// TwinCAT 3 PLC project Untitled1
// ProgramVersion: 3.1.4026.19
// libraries:
//   Tc2_Standard, * (Beckhoff Automation GmbH)
//   Tc2_System, * (Beckhoff Automation GmbH)
//   Tc2_Utilities, * (Beckhoff Automation GmbH)
//   Tc3_EventLogger, * (Beckhoff Automation GmbH)
//   Tc3_Module, * (Beckhoff Automation GmbH)
// project tree:
//   DUTs/ FlexChain.TcDUT, E_LightStates.TcDUT, E_SwitchType.TcDUT (not stored)
//   FaultChecker/ E_EventType.TcDUT, FB_EventTrigger.TcPOU, TriggerData.TcDUT, TC_EventSeverityToString.TcPOU, TriggerSettings.TcDUT
//   GVLs/ GVL_Fault.TcGVL, GVL_IO.TcGVL
//   Junk/ CdEventSeverity.TcTLEO, E_MachineStatus.TcDUT, FB_FaultChecker.TcPOU
//   / PlcTask.TcTTO
//   POUs/ fbDigitalInput.TcPOU, DigitalIO.TcPOU, fbDigitalOutput.TcPOU, MAIN.TcPOU
//   POUs/Hardware/PULS PISA/DTUs/ CircuitBreakerStatus.TcTLEO, PisaPulseCommMode.TcTLEO, PISA_HMI.TcDUT, PISA_IO.TcDUT, PulsPisaChannelCount.TcTLEO, TimedPulse.TcDUT
//   POUs/Hardware/PULS PISA/POUs/ FB_PISA.TcPOU, NTP.TcPOU
// real-time tasks:
//   TASK PlcTask: cycle T#2ms, priority 20, ADS port 350
// I/O:
//   DEVICE Device 1 (EtherCAT) (disabled), AmsNetId 10.1.14.1.2.1
//     Term 7 (EK1200)
//     Box 12 (Flexi Gateway GETC1)
//     Box 13 (EP6228-0022)
//   DEVICE Device 2 (EtherCAT), AmsNetId 0.0.0.0.3.1
//     Box 1 (EP6228-0022) [EP6228-0022 (IO Link Master)]
//       modules: Module 1 (DeviceState Inputs Device), Module 2 (DeviceState Inputs), Module 3 (empty), Module 4 (empty), Module 5 (empty), Module 6 (empty), Module 7 (empty), Module 8 (empty), Module 9 (empty), Module 10 (IO-Link Slave)
// variable links:
//   Untitled1/Untitled1 Instance <-> Device 1 (EtherCAT)/Box 13 (EP6228-0022)
//     PlcTask Inputs/GVL_IO.Encoder_Counts <-> Module 3 (IO-Link Slave)/IO-Link Port1/Counter
//     PlcTask Inputs/GVL_IO.flexChain.pdo[0] <-> Module 4 (IO-Link Slave)/IO-Link Port2_in/Process Data In
//     PlcTask Inputs/GVL_IO.flexChain.pdo[{1..12}] <-> Module 4 (IO-Link Slave)/IO-Link Port2_in/Process Data In_{1..12}  (12 links)
//   Untitled1/Untitled1 Instance <-> Device 1 (EtherCAT)/Term 7 (EK1200)/Term 10 (EL2008)
//     PlcTask Outputs/GVL_IO.aOutputs[1] <-> Channel 1/Output
//     PlcTask Outputs/GVL_IO.aOutputs[2] <-> Channel 2/Output
//   Untitled1/Untitled1 Instance <-> Device 1 (EtherCAT)/Term 7 (EK1200)/Term 9 (EL1008)
//     PlcTask Inputs/GVL_IO.aInputs[1] <-> Channel 1/Input
//     PlcTask Inputs/GVL_IO.aInputs[2] <-> Channel 2/Input
//     PlcTask Inputs/GVL_IO.aInputs[8] <-> Channel 8/Input
//   Untitled1/Untitled1 Instance <-> Device 2 (EtherCAT)/Box 1 (EP6228-0022)
//     PlcTask Inputs/MAIN.myPisa.PisaIO.bRX <-> Module 10 (IO-Link Slave)/IO-Link Port8_in/DI [X1.6-2] (pin 2)
//     PlcTask Outputs/MAIN.myPisa.PisaIO.bTX <-> Module 10 (IO-Link Slave)/IO-Link Port8_out/DO [X1.6-1] (pin 4)

CONFIGURATION Untitled1
    RESOURCE PLC ON TwinCAT3
        TASK PlcTask(INTERVAL := T#2ms, PRIORITY := 20);
        PROGRAM MAIN WITH PlcTask : MAIN;
    END_RESOURCE
END_CONFIGURATION

// ---- DUTs/FlexChain.TcDUT
TYPE FlexChain :
STRUCT
	pdo AT %I* : ARRAY[0..31] OF BYTE;//max pdo inputs of the flex chain bus
END_STRUCT
END_TYPE

// ---- DUTs/E_LightStates.TcDUT
{attribute 'qualified_only'}
{attribute 'strict'}
TYPE E_LightStates :
(
	OFF := 3,
	ON := 1,
	SLOW_BLINK := 2,
	FAST_BLINK := 0,
	
	
	COUNT  //Max value. Insert new values before to keep this as the max. Used to get max enum size when useful as an input to other function blocks.  
);
END_TYPE

// ---- FaultChecker/E_EventType.TcDUT
{attribute 'qualified_only'}
{attribute 'strict'}
{attribute 'to_string'}
TYPE E_EventType :
(
	Message := 0,
	Alarm :=1
);
END_TYPE

// ---- FaultChecker/TriggerData.TcDUT
TYPE TriggerData :
STRUCT
	nActivationCount: UDINT := 0;
	bTriggered : BOOL;
	
	GetEventTrigger : R_TRIG;
		

	timerDebounceTimer :TON;
	



	
	SendEventTrigger : R_TRIG;

END_STRUCT
END_TYPE

// ---- FaultChecker/TriggerSettings.TcDUT
TYPE TriggerSettings :
STRUCT
	//Settings
	tDebounceTime: TIME :=T#0S;
	nActivationThreshold: UDINT:=1;
	bAutoResetCount: BOOL :=TRUE;
	eEventType :E_EventType:=E_EventType.Message;
END_STRUCT
END_TYPE

// ---- Junk/CdEventSeverity.TcTLEO
{attribute 'qualified_only'}
{attribute 'strict'}
{attribute 'to_string'}
TYPE CdEventSeverity :
(
    Verbose:=0,     // Useful Information for debugging 
    Info:=1,        // Useful Information for operators
    Warning:=2,     // Machine operation not inhibited but at risk of becoming so
    Error:=3,       // Component operation blocked till resolved
    Critical:=4,    // Machine operation bloced till resolved
	                // 5-7 Reserved for future implementaion
	Lockout:=8      // Mackine locked out from use until ADMIN clears Fault 
					// 9 Reserved for future implementaion 
	
);
END_TYPE
//  Lockout = '8      '

// ---- Junk/E_MachineStatus.TcDUT
//{attribute 'qualified_only'}
//{attribute 'strict'}
{attribute 'to_string'}


(*
  |  1---    |  -2---   |  --3-    |   ---4   |  
 -+----------+----------+----------+----------+
0 | System   | Verbose  |    #     |     #    |
1 | Saftey   | Info     |    #     |     #    |
2 | Motor    | Warning  |    #     |     #    |
3 | Air      | Error    |    #     |     #    |
4 | Jam      | Critical |    #     |     #    |
5 | Heat     |          |    #     |     #    |
6 | Reject   |          |    #     |     #    |
7 | Fold     |          |    #     |     #    |
8 | Conveyor | Lockout  |    #     |     #    |
9 | General  |          |    #     |     #    |
  +----------+----------+----------+----------+
*)



TYPE E_MachineStatus:
(
	None                                := 0000,
	//System 0000-0999
	System_Standby		                := 0100,
	System_Running		                := 0101,
    System_Paused 		                := 0102,
	System_VFD_FirmwareUpdate           := 0199,
	Test_Mode           			    := 0104,
	Maintenance_Mode 	                := 0105,
	JogReverse 			                := 0106,
	System_FileError	                := 0400,
	
	//Safety 1000-1999	
	Reset_Safety	                    := 1101,	
	Safety_Fault	                    := 1401,
	Safety_System_Error	                := 1402,
	
	//Saftey - E-STOP XX10-XX19
	EStop_Triggered                     := 1410,
	Front_Left_ES                       := 1411,
	Front_Right_ES                      := 1412,
	Rear_Left_ES                        := 1413,
	Rear_Right_ES                       := 1414,
	External_ES                         := 1415,
	EStop_FB_Fault                     	:= 1419,
	
	//Saftey - Door XX20-XX29
	DoorOpen	                        := 1420,
	Top_Left_Door                       := 1421,
	Top_Right_Door                      := 1422,
	Left_Door                           := 1423,
	Right_Door                          := 1424,
	Rear_Door                           := 1425,
	Front_Panel                         := 1426,
	Door_FB_Fault                       := 1429,
	
	//Motor Fault 2000-2999	
	Skis_Calibrating                    := 2111,
	Motor_Fault	                        := 2450,
	VFD_Primary_Fault                   := 2451,
	VFD_XF1_Fault                       := 2452,
	VFD_XF2_Fault                       := 2453,
	VFD_Stacker_Fault                   := 2454,
	Inlet_Fault                         := 2455,
	Ski_Fault                           := 2456,
	Exit_1_Fault                        := 2461,
	Exit_2_Fault                        := 2462,
	Exit_3_Fault		                := 2463,
	Exit_4_Fault                        := 2464,
	Side_Conveyor_Fault                 := 2470,
	Side_Incline_Fault                  := 2471,
	Side_Conveyor_Unplugged             := 2472,
	
	VFD_Primary_Voltage_Loss            := 2180,
	VFD_XF1_Voltage_Loss                := 2181,
	VFD_XF2_Voltage_Loss                := 2182,
	VFD_Stacker_Voltage_Loss            := 2183,
	VFD_MultipleVoltage_Loss            := 2184,
	
	//Air Status 3000-3999	
	LowAirPressure	                    := 3120,
	HighAirWarning                      := 3221,
	LowAirWarning                       := 3220,
	Filter_Cleaning_Required            := 3333,
	
	//Jam Status 4000-4999	
	Jam_Detected		                := 4400,
	Jam_Inlet                           := 4401,
	Jam_Primary                         := 4402,
	Jam_XF1                             := 4403,
	Jam_XF2                             := 4404,
	Jam_XF2_SensorTimeout               := 4405,
	Jam_Stacker                         := 4406,
	Jam_Stacker_SensorTimeout           := 4407,
	Jam_Stacker_Lane1                   := 4408,
	Jam_Stacker_Lane2                   := 4409,
	Jam_Stacker_Lane3                   := 4410,	
	Jam_Stacker_Lane4                   := 4411,
	Jam_Reject_Rear                     := 4412, 	
	Jam_Reject_Front                    := 4413,
	Jam_Measure_Sensor                  := 4414,
	
	Jam_OverTorquePrimary               := 4415,
	Jam_OverTorqueXF1                   := 4416,
	Jam_OverTorqueXF2                   := 4417,
	Jam_OverTorqueStacker               := 4418,

	//Reject 6000-6999
	//Reject - USER XX00-XX09
	User_Reject                         := 6100,
	User_Reject_Damage                  := 6101,
	User_Reject_Tear  			        := 6102,
	User_Reject_Feed					:= 6103,
	User_Reject_Stain                   := 6104,
	//Reject - Auto XX10-xx40
	Auto_Reject_Unknown                 := 6111,
	OverWideL_Reject                    := 6112,
	OverWideR_Reject                    := 6113,
	Auto_Reject_TooNarrow               := 6114,
	Auto_Reject_TooWide                 := 6115,
	Auto_Reject_TooShort                := 6116,
	Auto_Reject_TooLong                 := 6117,
	Auto_Reject_WrongWidth              := 6118,
	Auto_Reject_WrongLength             := 6119,
	Auto_Reject_XF2_Timeout             := 6121,
	Auto_Reject_ConvLockout             := 6122,
	Auto_Reject_WrongSort               := 6123,
	Auto_Reject_Primary                 := 6124,
	Auto_Reject_Primary_NoSortNum       := 6125,
	Auto_Reject_Crossfold_1             := 6126,
	Auto_Reject_Crossfold_2             := 6127,
	Auto_Reject_Stacker                 := 6128,
	Reject_Unknown	                    := 6129,
		
	//Conveyor	
	Side_Conv_Full                      := 8102,
	Side_Conv_Top_Full 	                := 8103,
	
	//General
	Verbose                             := 9100,
	Info                                := 9200,
	Warning                             := 9300,
	Error                               := 9400,
	Critical                            := 9500,
	Lockout                             := 9800,
	//General - Circuit Breaker XX11-XX19
	Circuit_Breaker_Tripped             := 9411,
	Circuit_Breaker_Tripped_Repeat		:= 9421,
	Circuit_Breaker_Comms_Loss          := 9311,

	//General - SensorAllignment XX20-xx40
	MeasureSensorAlign	                := 9220,
	OverwideLSensorAlign                := 9221,				
	OverwideRSensorAlign                := 9222,
	XF1SensorAlign                      := 9223,
	XF2SensorAlign                      := 9224,
	Stack1SensorAlign                   := 9225, 
	Stack2SensorAlign                   := 9226,
	Stack3SensorAlign                   := 9227,
	Stack4SensorAlign                   := 9228,
	Sort1SensorAlign                    := 9229,
	Sort2SensorAlign                    := 9230,
	Sort3SensorAlign                    := 9231,
	Sort4SensorAlign                    := 9232,	
	Reserved                            := 9999//Leave as last so there aren't compile errors when copy pasting comma seperated values.
)INT;
END_TYPE

// ---- POUs/Hardware/PULS PISA/DTUs/CircuitBreakerStatus.TcTLEO
{attribute 'qualified_only'}
{attribute 'strict'}
TYPE CircuitBreakerStatus :
(
	OFF        := 0, // Channel has been set OFF either manually or programatically (only available in bidirectional mode)
	ON         := 1, // Channel is ON and funcioning normally (only available in bidirectional mode)
	TRIPPED    := 2, // An overcurrent event has tripped the device
	RESET      := 3, // A reset signal has been sent to the device but it hasn't responded yet
	UNKNOWN    := 4, // Comms isssue, data not yet recived, 
	NOTTRIPPED := 5  // Channel is OFF or ON (only available in unidirectional mode)  
);
END_TYPE

// ---- POUs/Hardware/PULS PISA/DTUs/PisaPulseCommMode.TcTLEO
{attribute 'qualified_only'}
{attribute 'strict'}
TYPE PisaPulseCommMode :
(
	Offline :=0,
	Unidirectional := 1,
	Bidirectional :=2
	
);
END_TYPE

// ---- POUs/Hardware/PULS PISA/DTUs/PISA_HMI.TcDUT
TYPE PISA_HMI :
STRUCT
	sCommMode : PisaPulseCommMode := PisaPulseCommMode.Offline;	
	//Variables for Reading
	aStatus : ARRAY[1..8] OF CircuitBreakerStatus := [8(CircuitBreakerStatus.UNKNOWN)];
	aTargetStatus : ARRAY[1..8] OF CircuitBreakerStatus := [8(CircuitBreakerStatus.UNKNOWN)];
END_STRUCT
END_TYPE

// ---- POUs/Hardware/PULS PISA/DTUs/PISA_IO.TcDUT
TYPE PISA_IO :
STRUCT
	sProductName  :STRING;
	bRX AT %I* : BIT;//INPUTS (STATUS -3.4)
	bTX AT %Q* : BIT;//OUTPUTS (CTRL +3.1)
END_STRUCT
END_TYPE

// ---- POUs/Hardware/PULS PISA/DTUs/PulsPisaChannelCount.TcTLEO
{attribute 'qualified_only'}
{attribute 'strict'}
TYPE PulsPisaChannelCount :
(
	FOUR := 4,
	EIGHT :=8
);
END_TYPE

// ---- POUs/Hardware/PULS PISA/DTUs/TimedPulse.TcDUT
TYPE TimedPulse :
STRUCT
	tLeadingGap: TIME   := T#0MS;
	tHighSignal: TIME := T#0MS;
	tTrailingGap: TIME:= T#0MS;
END_STRUCT
END_TYPE

// ---- GVLs/GVL_Fault.TcGVL
{attribute 'qualified_only'}
VAR_GLOBAL
	fbEventTrigger : FB_EventTrigger(TC_EVENT_CLASSES.TestEventClass); 
END_VAR

// ---- GVLs/GVL_IO.TcGVL
{attribute 'qualified_only'}

VAR_GLOBAL CONSTANT
    lightBarPDOstartIndex     : INT := 5;
    lightBarPDOsecondIndex : INT := lightBarPDOstartIndex+1;
END_VAR
VAR_GLOBAL
		Encoder_Counts AT %I* : UINT;
		
		byteArray AT %I* : ARRAY[1..8] OF BOOL;
		byteInt AT %I* : BYTE;
		flexChain : FlexChain;
		(*
		aLightCurtain AT %I* : ARRAY[1..10] OF POINTER TO BOOL := [flexChain.pdo[lightBarPDOstartIndex].0, 
																   flexChain.pdo[lightBarPDOstartIndex].1,
																   flexChain.pdo[lightBarPDOstartIndex].2,
																   flexChain.pdo[lightBarPDOstartIndex].3,
																   flexChain.pdo[lightBarPDOstartIndex].4,
																   flexChain.pdo[lightBarPDOstartIndex].5,
																   flexChain.pdo[lightBarPDOstartIndex].6,
																   flexChain.pdo[lightBarPDOstartIndex].7,
																   flexChain.pdo[lightBarPDOsecondIndex].0,
																   flexChain.pdo[lightBarPDOsecondIndex].1];
																   
																   *)
																   

END_VAR

// ---- POUs/MAIN.TcPOU
PROGRAM MAIN

VAR
	

	
	bGreenBtn    : POINTER TO BOOL:= ADR(GVL_IO.aInputs[1]);
	bRedBtn		: POINTER TO BOOL:= ADR(GVL_IO.aInputs[2]);
	bLight : POINTER TO BOOL := ADR(GVL_IO.aOutputs[1]);

	fbStartInput : fbDigitalInput(ioBitRef := ADR(GVL_IO.aInputs[1]), switchType := E_SwitchType.NO);
	fbStopInput : fbDigitalInput(ioBitRef := ADR(GVL_IO.aInputs[2]), switchType := E_SwitchType.NC);
	fbLightOutput : fbDigitalOutput(ioBitRef := ADR(GVL_IO.aOutputs[1]), switchType := E_SwitchType.NO);
	light2 : fbDigitalOutput(ioBitRef := ADR(GVL_IO.aOutputs[2]), switchType := E_SwitchType.NO);
	CurrentState: UINT  := TO_UINT(E_LightStates.FAST_BLINK);
	
	fbCounter : CTU;

	timedLight : BOOL;
	timer :TON;

	aLightCurtain : ARRAY[1..10] OF BOOL; 
	
	//myPisa : FB_PISA_Comms(sProductName := 'PISA-M-4CL2');

	cbStates : ARRAY[1..4] OF CircuitBreakerStatus;

	
	
	
	
	myPisa : FB_PISA(eChannelCount := PulsPisaChannelCount.Four, sDeviceName:= 'PULS PISA-M-4CL2');
	i: INT;
	aCurrentStates : ARRAY[1..4] OF CircuitBreakerStatus;
	aTargetStates : ARRAY[1..4] OF CircuitBreakerStatus := [4(CircuitBreakerStatus.UNKNOWN)];
	
	bRun : BOOL :=TRUE;
	bWrite: BOOL :=FALSE;
	status: PisaPulseCommMode;
	
	test: BOOL :=FALSE;
	
	bOnce :BOOL :=TRUE;
	fbFaultChecker : FB_FaultChecker;
	
	bTestTrigger1:BOOL:=FALSE;
	bTestTrigger2:BOOL:=FALSE;
	bTestTrigger3:BOOL:=FALSE;
	
	stDelayedActivation : TriggerSettings;
	stRepeatActivation : TriggerSettings;				   
					  

	
	nLastEventCount: UINT;
	nIndex: INT;
	in:UINT;
	//event: FB_FaultEvent;
	fbMessage : FB_TCMessage;
	bTest2: BOOL;
END_VAR

(*IF bOnce THEN
(*
event1:= FB_FaultEvent(bChannelOneTripped,
	                   tActivationDelay:=T#2S,
					   nActivationCount:=1,
					   sErrorName:='Circuit Breaker Tripped',
                       sErrorDescription:='Lane 1 conveyor motor over current. Check Tension',
					   eSeverity:=TcEventSeverity.Error);
*)

//fb_EventTrigger3.Activate(bBoolA :=FALSE);

//fbFaultChecker.AddTrigger(ADR(fb_eventTrigger1));
 // fbFaultChecker.AddTrigger(ADR(fb_eventTrigger2));

  fbFaultChecker.AddTrigger(ADR(fb_EventTrigger3));
  
bOnce := FALSE;
END_IF
*)
//TC_EVENTS.TestEventClass.TestEvent2.nEventId
stDelayedActivation.tDebounceTime:=T#3S;
stRepeatActivation.nActivationThreshold:=2;


GVL_Fault.fbEventTrigger.Configure(nEventID:=TC_EVENTS.TestEventClass.TestEvent1.nEventId,stDelayedActivation);
GVL_Fault.fbEventTrigger.Configure(nEventID:=TC_EVENTS.TestEventClass.TestEvent2.nEventId,stRepeatActivation);

GVL_Fault.fbEventTrigger.TriggerEvent(nEventEntry:=TC_EVENTS.TestEventClass.TestEvent1, bTestTrigger1,sSource:=__POUNAME());
GVL_Fault.fbEventTrigger.Trigger(nEventID:=TC_EVENTS.TestEventClass.TestEvent2.nEventId, bTestTrigger2);

TestSourceMethod();
//IF bTestTrigger1 THEN
	
//END_IF

(*
IF bChannelOneTripped THEN
	//fbMessage.CreateEx(TC_EVENTS.EventClass.Event,0);
	fbMessage.Create(eventClass:= 
END_IF
*)





fbFaultChecker();//update

myPisa(bEnable:=bRun, bBidirectional:=bWrite);



IF bTest2 THEN
	//myPisa.ResetAll();
ELSE	
//	FOR i := 1 TO 4 DO
//    	myPisa.SetStatus(nChannel:=i , eStatus:=aTargetStates[i]);
//	END_FOR;
END_IF

FOR i := 1 TO 4 DO
    aCurrentStates[i] := myPisa.GetStatus(i);
END_FOR;






status := myPisa.GetCommMode();


//bTestTrigger3:=status = PisaPulseCommMode.Offline;

GVL_IO.aOutputs[8] := GVL_IO.aInputs[8]; // Output 8 mirrors input 8





IF fbFaultChecker.GetActiveEventCount()<> nLastEventCount and test THEN
(*
FOR in := 0 TO fbFaultChecker.GetTotalEventCount()-1DO
	//fbFaultChecker.GetEvent(nIndex:=in)^.Active;
	
	
	IF (fbFaultChecker.GetEvent(nIndex:=in)^.GetState())THEN 
		ADSLOGSTR(
			msgCtrlMask := ADSLOG_MSGTYPE_HINT, 
			msgFmtStr   := fbFaultChecker.GetEvent(nIndex:=in)^.GetLongMessage(),
			strArg      := '');
	END_IF
END_FOR
*)
(*
ADSLOGSTR(
	msgCtrlMask := ADSLOG_MSGTYPE_HINT, 
	msgFmtStr   := fbFaultChecker.GetFirstActiveEvent()^.GetLongMessage(),
	strArg      := TO_STRING(fbFaultChecker.GetFirstActiveEvent()^.GetEventSeverity())
);


*)      
	nLastEventCount:=fbFaultChecker.GetActiveEventCount();
END_IF





























IF fbStartInput.Get() THEN
		fbLightOutput.Set(TRUE);
ELSE 
		fbLightOutput.Set(FALSE);
END_IF

//bGreenBtn := aInputs[1];


(*
IF bGreenBtn^ THEN
		bLight^:=TRUE;
ELSE 
		bLight^:=FALSE;
END_IF
*)




fbCounter(CU:=fbStartInput.Get(),CU:=fbStartInput.Get(), RESET :=fbStopInput.Get() ,PV := UINT_TO_WORD(E_LightStates.COUNT));
CurrentState:=fbCounter.CV;


	aLightCurtain[1]:= (GVL_IO.flexChain.pdo[GVL_IO.lightBarPDOstartIndex] AND 2#0000_0000_0000_0001) <> 0;
	aLightCurtain[2]:= (GVL_IO.flexChain.pdo[GVL_IO.lightBarPDOstartIndex] AND 2#0000_0000_0000_0010) <> 0;
	aLightCurtain[3]:= (GVL_IO.flexChain.pdo[GVL_IO.lightBarPDOstartIndex] AND 2#0000_0000_0000_0100) <> 0;
	aLightCurtain[4]:= (GVL_IO.flexChain.pdo[GVL_IO.lightBarPDOstartIndex] AND 2#0000_0000_0000_1000) <> 0;
	aLightCurtain[5]:= (GVL_IO.flexChain.pdo[GVL_IO.lightBarPDOstartIndex] AND 2#0000_0000_0001_0000) <> 0;
	aLightCurtain[6]:= (GVL_IO.flexChain.pdo[GVL_IO.lightBarPDOstartIndex] AND 2#0000_0000_0010_0000) <> 0;
	aLightCurtain[7]:= (GVL_IO.flexChain.pdo[GVL_IO.lightBarPDOstartIndex] AND 2#0000_0000_0100_0000) <> 0;
	aLightCurtain[8]:= (GVL_IO.flexChain.pdo[GVL_IO.lightBarPDOstartIndex] AND 2#0000_0000_1000_0000) <> 0;
	aLightCurtain[9]:= (GVL_IO.flexChain.pdo[GVL_IO.lightBarPDOsecondIndex] AND 2#0000_0000_0000_0001) <> 0;
	aLightCurtain[10]:= (GVL_IO.flexChain.pdo[GVL_IO.lightBarPDOsecondIndex] AND 2#0000_0000_0000_0010) <> 0;
								


CASE CurrentState OF
    E_LightStates.OFF:
		fbLightOutput.Set(FALSE);
    E_LightStates.ON:
		fbLightOutput.Set(TRUE);
    E_LightStates.SLOW_BLINK:
		timer(IN := NOT timer.Q, PT := T#1S500MS);
		IF timer.Q THEN 
			timedLight := NOT timedLight; 
		END_IF
		fbLightOutput.Set(timedLight);
    E_LightStates.FAST_BLINK:
		timer(IN := NOT timer.Q, PT := T#0S500MS);
		IF timer.Q THEN 
			timedLight := NOT timedLight; 
		END_IF
		fbLightOutput.Set(timedLight);
ELSE
		fbLightOutput.Set(FALSE);
		fbCounter(RESET:=TRUE);
		
END_CASE

IF GVL_IO.Encoder_Counts > 500 THEN
	light2.Set(TRUE);
ELSE
	light2.Set(FALSE);		

END_IF

METHOD TestSourceMethod
VAR
	source :FB_TcSourceInfo();
END_VAR

//.ResetToDefault();
//source.sName:=__CURRENT_FILE_NAME;

//GVL_Fault.fb_eventTrigger1.Activate(nEventID:=555,bTrigger:=bTestTrigger1, sSource:=__POUNAME());
GVL_Fault.fbEventTrigger.Trigger(nEventID:=555,bTrigger:=bTestTrigger3, sSource:=__POUNAME(),'2', '4','TRIPPED',eSeverity:=TcEventSeverity.Critical);
END_METHOD

END_PROGRAM

// ---- POUs/fbDigitalInput.TcPOU
FUNCTION_BLOCK fbDigitalInput EXTENDS fbDigitalIO

END_FUNCTION_BLOCK

// ---- POUs/fbDigitalOutput.TcPOU
FUNCTION_BLOCK fbDigitalOutput EXTENDS DigitalIO

METHOD PUBLIC Set
VAR_INPUT
	bValue : BOOL;
END_VAR
ioBIT^ := bValue;
END_METHOD

END_FUNCTION_BLOCK

// ---- POUs/DigitalIO.TcPOU
FUNCTION_BLOCK DigitalIO
VAR
	ioBIT : POINTER TO BOOL;
	bFakeValue : BOOL;
	bOverwriteEnable : BOOL;
	eSwitchType : E_SwitchType;
END_VAR

METHOD PUBLIC ClearOverride
VAR_INPUT
END_VAR
bOverwriteEnable := FALSE;
END_METHOD

METHOD FB_init : BOOL
VAR_INPUT
	bInitRetains : BOOL; // if TRUE, the retain variables are initialized (warm start / cold start)
	bInCopyCode : BOOL;  // if TRUE, the instance afterwards gets moved into the copy code (online change)
	ioBitRef : POINTER TO BOOL;
	switchType : E_SwitchType := E_SwitchType.NO; // No default :(
END_VAR
ioBIT := ioBitRef;
eSwitchType := switchType;
END_METHOD

METHOD PUBLIC Get : BOOL
IF bOverwriteEnable = TRUE THEN
	Get:= bFakeValue;
ELSE
	IF eSwitchType = E_SwitchType.NO THEN
		Get := ioBIT^;
	ELSIF eSwitchType = E_SwitchType.NC THEN
		Get := NOT ioBIT^;
	ELSE
		Get := ioBIT^;//TODO ERROR
	END_IF;
END_IF;
END_METHOD

METHOD PUBLIC GetRawValue : BOOL
GetRawValue := ioBIT^;
END_METHOD

METHOD PUBLIC GetSwitchType : E_SwitchType
VAR_INPUT
END_VAR
GetSwitchType := eSwitchType;
END_METHOD

METHOD PUBLIC SetOverride
VAR_INPUT
END_VAR
bOverwriteEnable := TRUE;
END_METHOD

END_FUNCTION_BLOCK

// ---- POUs/Hardware/PULS PISA/POUs/FB_PISA.TcPOU
FUNCTION_BLOCK FB_PISA
VAR_INPUT
	 bEnable	: BOOL; //When TRUE devices channel states will be read from device and stored for retreval by GetSatus()
	 bBidirectional	: BOOL; //When TRUE and bEnable target channel states as configured by SetStatus() will be sent to the device 
END_VAR
VAR CONSTANT
	//Constants as defined in Pulse Pisa Manuals
    MAX_NUMBER_OF_CHANNELS : USINT            := 8; //Theoritical max channels offered by Pulse is 64. Setting to 8 for now as we are unlikely to go beyond 8
	STANDARD_NUMBER_OF_CHANNELS : USINT       := 4;  
	
	SHORT_START_PULSE_DURATION : TIME := T#150MS;
	LONG_START_PULSE_DURATION : TIME  := T#200MS;
	
	DRIFT_TOLERANCE : TIME        := T#15MS;
	STATUS_DURATION: TIME         := T#100MS;
	STATUS_PERIOD_DURATION: TIME  := T#200MS;
	
	FOUR_CHANNEL_SEQUENCE_TIME :TIME := T#1100MS;
	EIGHT_CHANNEL_SEQUENCE_TIME :TIME := T#2200MS;
	
	WRITE_PERIODS_AFTER_DATA : USINT :=2;
	
	MIN_PULSE_DURATION: TIME     := T#50MS;	
	
END_VAR

VAR
	PisaIO : PISA_IO; // Struct for mapping PLC to physical IO Hardware
	PisaHMI : PISA_HMI; //Struct for mapping PLC to HMI
	
	lastPisaHMI : PISA_HMI; //Struct for latching states
	
	tWatchdogTime: TIME;
	timerReadSequenceWatchdog : TOF;
	
	bWriteRequestedHMI : BOOL;

	
	bStartBitFound : BOOL;//Indicateds the falling edge of the start bit has been found. (we are reading channels)
	nReadingChannelIndex	: USINT := 0 ; //The current channel number as determined by time or falling edges in the data
	nLastReadingChannelIndex :USINT :=0; //A lag behind value of the channel for correct array index because saving of channel data happends in the first time slice of the next channel 
	nNumberOfChannels : USINT := STANDARD_NUMBER_OF_CHANNELS;
	tLastPulseDuration : TIME; //Store the elapsed time. 
	
	timerPulseMeasurement :TON;
	timerReadPeriodMax : TP;
	timerPeriodMin :TON;
		
	inputFallingEdge: F_TRIG;
	maxTime: F_TRIG;//Indicates the maximum time of a channel has been hit
	bResetMaxTimeFlag: BOOL:=FALSE; //Used to indicate the max pulse timer needs to be reset NEXT cycle. Can't happen this cycle or Q will not trigger. 

	//Variables for Writing
	aCtrl : ARRAY[0..MAX_NUMBER_OF_CHANNELS+WRITE_PERIODS_AFTER_DATA] OF TimedPulse:= [(MAX_NUMBER_OF_CHANNELS+WRITE_PERIODS_AFTER_DATA)(sOnSignal)];
		
	timerLeadingGap : NTP; //TODO-NIKO See if this can be better rewritten to no use my strange extended timer. Or clean up the timer. should add unit test first as changing it breaks functionality currently
	timerWriteHigh : NTP;
	timerTrailingGap: NTP;
	
	fTimer1Done : F_TRIG;
	fTimer2Done : F_TRIG;
	fTimer3Done : F_TRIG;

	nNextWriteChannelFlag : BOOL:=TRUE;
	nWriteIndex : USINT;

	nDoneCount:USINT:=0;	
	nTimersToComplete: USINT :=0;

	//Command Durations	
	tGapTimeAdjustment :TIME:=T#5MS; //Needed to account for drift due to syscle time
    sStartBitSignal : TimedPulse := (tLeadingGap := T#000MS, tHighSignal := T#150MS, tTrailingGap := T#000MS);
	sResetSignal    : TimedPulse := (tLeadingGap := T#100MS - tGapTimeAdjustment, tHighSignal := T#100MS, tTrailingGap := T#000MS);
	sOnSignal       : TimedPulse := (tLeadingGap := T#200MS - tGapTimeAdjustment, tHighSignal := T#000MS, tTrailingGap := T#000MS);
	sOffSignal      : TimedPulse := (tLeadingGap := T#100MS - tGapTimeAdjustment, tHighSignal := T#050MS, tTrailingGap := T#050MS);
	sStopBitSignal  : TimedPulse := (tLeadingGap := T#100MS, tHighSignal :=T#100MS, tTrailingGap := T#050MS);
	sWaitBitSignal  : TimedPulse := (tLeadingGap := T#500MS, tHighSignal := T#000MS, tTrailingGap := T#000MS);
	
	nResetChannel :USINT:=1;
	
	timerResetDelay : TON;

	

	i: INT;
END_VAR

(*
//*****************************************************************Notes**********************************************************\\
Function Block for reading and writing channel states to PULS PISA line of smart circuit breaker products.
https://products.pulspower.com/us/product-families/pisa.html

Implemented and tested at 2MS Cycle Time. Different Cycle times could cause communication issues with device. 
10MS cycle time may be suficient for reading but the software on the PISA-M will not interpret written signals correctly at +/-10MS
Code was written with to accomidate for different numbers of device channels but has only been tested with the the 4 channel PISA-M-4CL2
 
//*****************************************************************Revs**********************************************************\\
   (          who            )(    Date    ) (   Rev     ) (								Disc						)
     Nikolas Gamarra		 	2025.09.26		1.0.0		Initial Code
	
//*****************************************************************Code**********************************************************\\
*)
IF bEnable THEN
	
	ReadFromDevice();
	
	bWriteRequestedHMI:=FALSE;
	
	
	
	
	

	
	
	IF bBidirectional THEN
		
	
		FOR i := 1 TO nNumberOfChannels DO
		IF PisaHMI.aStatus[i] = CircuitBreakerStatus.OFF AND lastPisaHMI.aStatus[i] = CircuitBreakerStatus.ON AND PisaHMI.aTargetStatus[i] = CircuitBreakerStatus.ON THEN
			PisaHMI.aTargetStatus[i] := CircuitBreakerStatus.OFF; 
		END_IF
		IF PisaHMI.aStatus[i] = CircuitBreakerStatus.ON AND lastPisaHMI.aStatus[i] = CircuitBreakerStatus.OFF AND PisaHMI.aTargetStatus[i] = CircuitBreakerStatus.OFF THEN
			PisaHMI.aTargetStatus[i] := CircuitBreakerStatus.ON; 
		END_IF
		
		IF PisaHMI.aStatus[i] = lastPisaHMI.aStatus[i] AND PisaHMI.aTargetStatus[i] <> lastPisaHMI.aTargetStatus[i] THEN
			bWriteRequestedHMI:=TRUE;
		END_IF
		
		
	END_FOR
	
		
		WriteToDevice();
	ELSE
		ResetWriteIndex();
		CopyReadValuesToTargetValues();
	END_IF	
	
	lastPisaHMI:= PisaHMI;
ELSE// Program not running.
	ClearStatus();
	ClearTarget();
END_IF

METHOD PRIVATE ClearStatus
VAR_INPUT
END_VAR
VAR
	i : INT;//array index
END_VAR
FOR i := 1 TO nNumberOfChannels DO
	// Wipe out the array. 	
	PisaHMI.aStatus[i] := CircuitBreakerStatus.UNKNOWN; 
END_FOR
END_METHOD

METHOD PRIVATE ClearTarget
VAR_INPUT
END_VAR

VAR
	i: INT;
END_VAR
FOR i := 1 TO nNumberOfChannels DO
	// Wipe out the array 	
	PisaHMI.aTargetStatus[i] := CircuitBreakerStatus.UNKNOWN;
END_FOR
END_METHOD

METHOD PRIVATE CopyReadValuesToTargetValues
VAR_INPUT
END_VAR

VAR
	i: INT;
END_VAR
FOR i := 1 TO nNumberOfChannels DO
    PisaHMI.aTargetStatus[i] := PisaHMI.aStatus[i];
END_FOR;
END_METHOD

METHOD FB_init : BOOL
VAR_INPUT
	bInitRetains : BOOL; // if TRUE, the retain variables are initialized (warm start / cold start)
	bInCopyCode : BOOL;  // if TRUE, the instance afterwards gets moved into the copy code (online change)
	eChannelCount : PulsPisaChannelCount;// Number of independent circuit breaker channels on the device
	sDeviceName: STRING;// Name of the device for reference later when building error messages
END_VAR
aCtrl[0]:=sStartBitSignal;
aCtrl[nNumberOfChannels+1]:=sStopBitSignal;
nNumberOfChannels := TO_USINT(eChannelCount);

PisaIO.sProductName:=sDeviceName;

IF eChannelCount = PulsPisaChannelCount.Eight THEN
	tWatchdogTime:=EIGHT_CHANNEL_SEQUENCE_TIME ;
ELSE
	tWatchdogTime:=FOUR_CHANNEL_SEQUENCE_TIME ;
END_IF
END_METHOD

METHOD PUBLIC GetChannelCount : USINT
VAR_INPUT
END_VAR
GetChannelCount := nNumberOfChannels;
END_METHOD

METHOD PUBLIC GetCommMode : PisaPulseCommMode //The current operational mode of the device
GetCommMode:=PisaHMI.sCommMode;
END_METHOD

METHOD PUBLIC GetDeviceName : STRING
GetDeviceName:=PisaIO.sProductName;
END_METHOD

METHOD GetStatus : CircuitBreakerStatus // The state of provided channel
VAR_INPUT
	nChannel : UINT; // The device channel to check the state of
END_VAR
IF nChannel > 0 AND nChannel <= nNumberOfChannels THEN
	GetStatus := PisaHMI.aStatus[nChannel];
ELSE
	GetStatus := CircuitBreakerStatus.UNKNOWN;
END_IF
END_METHOD

METHOD PRIVATE ReadFromDevice : BOOL
VAR_INPUT
END_VAR
timerPulseMeasurement(IN := PisaIO.bRX , PT:=tWatchdogTime);
	

inputFallingEdge(CLK := PisaIO.bRX);//Indicates any falling edge on the input signal 
maxTime(CLK:= timerReadPeriodMax.Q);//Indicates the max period time has elapsed

IF bResetMaxTimeFlag THEN
	timerReadPeriodMax(IN:=TRUE);
	bResetMaxTimeFlag :=FALSE;
ELSE
	timerReadPeriodMax(IN:=inputFallingEdge.Q AND NOT timerReadPeriodMax.Q, PT:= STATUS_PERIOD_DURATION);
END_IF

IF( PisaIO.bRX = TRUE AND NOT inputFallingEdge.Q AND NOT timerPulseMeasurement.Q) THEN // IF the input is high, update the running counter of the pulse duration
	tLastPulseDuration := timerPulseMeasurement.ET;	
END_IF

timerReadSequenceWatchdog(IN := inputFallingEdge.Q, PT:= tWatchdogTime);

IF (timerReadSequenceWatchdog.Q = FALSE) THEN//Our watchdog has expired
	PisaHMI.sCommMode := PisaPulseCommMode.Offline;	
	ClearStatus();
END_IF

IF (inputFallingEdge.Q)THEN //A pulse just completed

	
	IF tLastPulseDuration >= SHORT_START_PULSE_DURATION - DRIFT_TOLERANCE THEN
		IF tLastPulseDuration >= T#155MS(*LONG_START_PULSE_DURATION - DRIFT_TOLERANCE THEN*) THEN
			PisaHMI.sCommMode := PisaPulseCommMode.Unidirectional;
		ELSE
			PisaHMI.sCommMode := PisaPulseCommMode.Bidirectional;
		END_IF
		
		bStartBitFound 	:= NOT bStartBitFound; // Main reset happens elsewhere. Failsafe here. Only happense every other cycle but acceptable as only a failsafe.
		ResetReadIndex();//Reset counter to prepair for next cycle 
		tLastPulseDuration :=T#0MS ;// reset the time counter so we can measure next pulses
		
	END_IF
END_IF

IF (((maxTime.Q = TRUE AND PisaIO.bRX = FALSE )) AND bStartBitFound = TRUE) THEN 
	IF timerPeriodMin.Q THEN
		nReadingChannelIndex := nReadingChannelIndex + 1;
		timerPeriodMin(IN:= FALSE, PT:=DRIFT_TOLERANCE);
	END_IF 
ELSE
	timerPeriodMin(IN:= TRUE, PT:=DRIFT_TOLERANCE);			
END_IF

IF bStartBitFound THEN // Only calculate state if we have found the start bit and thus are in the channel bits
	IF (nLastReadingChannelIndex <> nReadingChannelIndex) THEN//We have advanced to the gap period after a readin of a pulse
		
		bResetMaxTimeFlag:=TRUE;

		IF tLastPulseDuration >= DRIFT_TOLERANCE THEN //have a positive signal
			IF tLastPulseDuration >= MIN_PULSE_DURATION - DRIFT_TOLERANCE THEN //Signal large enough than smallest expected
				IF tLastPulseDuration > STATUS_DURATION - DRIFT_TOLERANCE THEN
					PisaHMI.aStatus[nLastReadingChannelIndex]	:= CircuitBreakerStatus.TRIPPED;
				ELSIF tLastPulseDuration > MIN_PULSE_DURATION - DRIFT_TOLERANCE THEN
					PisaHMI.aStatus[nLastReadingChannelIndex]	:= CircuitBreakerStatus.OFF;
				ELSE //should never happen
					ClearStatus();
				END_IF	
			ELSE//Likely indicates out of sync
				ClearStatus();
			END_IF
		ELSE
			IF PisaHMI.sCommMode = PisaPulseCommMode.Bidirectional THEN	
				PisaHMI.aStatus[nLastReadingChannelIndex]	:= CircuitBreakerStatus.ON;
			ELSE
				PisaHMI.aStatus[nLastReadingChannelIndex]	:= CircuitBreakerStatus.NOTTRIPPED;
			END_IF
		END_IF
				
		tLastPulseDuration :=T#0MS ;// reset the time counter as we have recorded the measurement for this pulse
		nLastReadingChannelIndex := nReadingChannelIndex;
	END_IF

	IF nReadingChannelIndex > nNumberOfChannels THEN //End of Sequence
		bStartBitFound := FALSE;
	END_IF
END_IF
END_METHOD

METHOD PRIVATE ResetAll // Sequencial rolling reseet of all channels
timerResetDelay(IN:= NOT timerResetDelay.Q,PT:=tWatchdogTime );

IF timerResetDelay.Q THEN
	nResetChannel :=nResetChannel+1;
END_IF

//Perform a rolling reseet of all channels. (off by 1 index is ok a setter rejects out of bounds args)
SetStatus(nChannel:=nResetChannel, eStatus:=CircuitBreakerStatus.RESET);
SetStatus(nChannel:=nResetChannel-1, eStatus:=CircuitBreakerStatus.ON);


IF nResetChannel > nNumberOfChannels THEN
	nResetChannel:=1;
END_IF
END_METHOD

METHOD PRIVATE ResetReadIndex
nReadingChannelIndex :=1;
nLastReadingChannelIndex:=1;
END_METHOD

METHOD PRIVATE ResetWriteIndex
PisaIO.bTX:=FALSE;
nNextWriteChannelFlag:=TRUE;
nWriteIndex:=0;	
aCtrl[0]:=sStartBitSignal;
aCtrl[nNumberOfChannels+1]:=sStopBitSignal;
aCtrl[nNumberOfChannels+2]:=sWaitBitSignal;
END_METHOD

METHOD SetStatus
VAR_INPUT
	nChannel : UINT; // The device channel to change
	eStatus : CircuitBreakerStatus; // The desired stat to change to
END_VAR
IF nChannel >0 AND nChannel<=nNumberOfChannels THEN
	PisaHMI.aTargetStatus[nChannel]:=eStatus;//Actual settingof the desired status to device
	IF (PisaHMI.aStatus[nChannel] <> CircuitBreakerStatus.ON)THEN//Fake a status of reset but only if the device hasn't yet successfully reset
		IF(eStatus = CircuitBreakerStatus.RESET AND PisaHMI.sCommMode =  PisaPulseCommMode.Bidirectional)  THEN
			PisaHMI.aStatus[nChannel] := CircuitBreakerStatus.RESET;
		END_IF
	END_IF
END_IF
END_METHOD

METHOD PRIVATE WriteToDevice : BOOL
VAR_INPUT
END_VAR
IF nNextWriteChannelFlag THEN
	nTimersToComplete:=0;
	IF(aCtrl[nWriteIndex].tLeadingGap > T#0MS)THEN
		nTimersToComplete:=nTimersToComplete+1;
	END_IF
	IF(aCtrl[nWriteIndex].tHighSignal > T#0MS)THEN
		nTimersToComplete:=nTimersToComplete+1;
	END_IF
	IF(aCtrl[nWriteIndex].tTrailingGap > T#0MS)THEN
		nTimersToComplete:=nTimersToComplete+1;
	END_IF
END_IF

timerLeadingGap(IN:=nNextWriteChannelFlag, PT:=aCtrl[nWriteIndex].tLeadingGap);
timerWriteHigh(IN:= NOT timerLeadingGap.Q AND NOT nNextWriteChannelFlag, PT:=aCtrl[nWriteIndex].tHighSignal);
timerTrailingGap(IN:= NOT timerWriteHigh.Q AND NOT timerWriteHigh.Q AND NOT nNextWriteChannelFlag AND nDoneCount>0, PT:=aCtrl[nWriteIndex].tTrailingGap);

fTimer1Done(CLK:= timerLeadingGap.Q);
fTimer2Done(CLK:= timerWriteHigh.Q);
fTimer3Done(CLK:= timerTrailingGap.Q);


IF (fTimer1Done.Q OR  fTimer2Done.Q OR fTimer3Done.Q)AND NOT nNextWriteChannelFlag THEN
	nDoneCount := nDoneCount +1;
END_IF


nNextWriteChannelFlag:=FALSE;
IF nDoneCount >= nTimersToComplete  THEN

	nDoneCount:=0;
	nWriteIndex := nWriteIndex + 1;
	nNextWriteChannelFlag:=TRUE;
	
	
	IF(nWriteIndex>0 AND nWriteIndex <nNumberOfChannels+1) THEN
		//Update any target values. Won't execute till next cycle
		CASE PisaHMI.aTargetStatus[nWriteIndex] OF 
		CircuitBreakerStatus.OFF, CircuitBreakerStatus.TRIPPED:
			aCtrl[nWriteIndex]:=sOffSignal;
		CircuitBreakerStatus.On, CircuitBreakerStatus.NOTTRIPPED:
			aCtrl[nWriteIndex]:=sOnSignal;
		CircuitBreakerStatus.RESET :
			aCtrl[nWriteIndex]:=sResetSignal;
		ELSE // Default (UNKNOWN)
			//replace the unknown with the read value
			PisaHMI.aTargetStatus[nWriteIndex] := PisaHMI.aStatus[nWriteIndex];
			//repeat this step
			nDoneCount:=99;
			nWriteIndex:=nWriteIndex-1;
			
			
			//aCtrl[nWriteIndex]:=sOnSignal;
		END_CASE;
	END_IF	
END_IF

IF(nWriteIndex >nNumberOfChannels + WRITE_PERIODS_AFTER_DATA) THEN  
		ResetWriteIndex();
END_IF

PisaIO.bTX:=timerWriteHigh.Q;//Write to digital output
END_METHOD

END_FUNCTION_BLOCK

// ---- POUs/Hardware/PULS PISA/POUs/NTP.TcPOU
FUNCTION_BLOCK NTP EXTENDS TP
VAR_INPUT
END_VAR
VAR_OUTPUT
	bDone: BOOL;
END_VAR
VAR
	timer :TP;
	bHasBeenStarted :BOOL :=FALSE;
	//(IN:= NOT timerWriteLow.Q AND NOT bNextFlag, PT:=aCtrl[nWriteIndex].tHigh);
	//fbWriteQFalling(clk:=timerWriteHigh.Q);
END_VAR

IF PT = T#0MS THEN
	Q := FALSE;
	bDone:=TRUE;
ELSE
	timer(IN:= IN, PT:= PT);
	ET:=timer.ET;
	Q:=timer.Q;
	
	IF(IN = TRUE)THEN 
		bHasBeenStarted:=TRUE;
	END_IF
	IF bDone THEN
		bHasBeenStarted:=FALSE;
	END_IF
	
	
	bDone:= NOT timer.Q AND bHasBeenStarted;
	//TODO-NIKO Remove local timer and call super? Needs testing, wasn't behaving as expected.
	//SUPER^.IN:=IN;
	//SUPER^.PT:=PT;	
	//Q := SUPER^.Q;
	//ET:= SUPER^.ET;

END_IF

METHOD PUBLIC Reset : BOOL
VAR_INPUT
END_VAR
bHasBeenStarted:=FALSE;
bDone:=FALSE;
END_METHOD

END_FUNCTION_BLOCK

// ---- Junk/FB_FaultChecker.TcPOU
FUNCTION_BLOCK FB_FaultChecker
VAR_INPUT
END_VAR
VAR_OUTPUT
END_VAR
VAR_IN_OUT
    //aFaultsToCheck  : ARRAY [*] OF POINTER TO FB_FaultEvent;
	
END_VAR
VAR CONSTANT
	//Constants as defined in Pulse Pisa Manuals
    MAX_FAULTS : USINT            := 255;     
END_VAR

VAR
	
aFaultsToCheck : ARRAY[0..MAX_FAULTS] OF POINTER TO FB_EventTrigger;
	//aFaultsToCheck  : ARRAY [255] OF POINTER TO FB_FaultEvent;
	nIdx   : DINT;
    nSum   : DINT;
	nWriteIndex :UINT:=0;
	nLastWriteIndex:UINT:=0;
	
	
	//aFaultsToCheck : ARRAY[1..MAX_NUMBER_OF_CHANNELS] OF CircuitBreakerStatus := [MAX_NUMBER_OF_CHANNELS(CircuitBreakerStatus.UNKNOWN)]; 
	fbFaultChecker: INT;
	bTest: BOOL :=FALSE;
	bFlag : BOOL;
	timerDelay : TOF;
	

END_VAR

Update();

METHOD PUBLIC AddTrigger
VAR_INPUT
	fbEvent : POINTER TO FB_EventTrigger;
END_VAR

aFaultsToCheck[nWriteIndex]:=fbEvent;
nWriteIndex := nWriteIndex +1;
END_METHOD

METHOD GetActiveEventCount : UINT
VAR
	nActiveEventCount:UINT:=0;
END_VAR
//FOR nIdx := LOWER_BOUND(aFaultsToCheck,1) TO UPPER_BOUND(aFaultsToCheck,1) DO

FOR nIdx := 0 TO nWriteIndex-1 DO
	//IF(aFaultsToCheck[nIdx]^.GetState())THEN
		//nActiveEventCount:=nActiveEventCount+1;
///	END_IF
END_FOR;
GetActiveEventCount:=nActiveEventCount;
END_METHOD

METHOD PUBLIC GetEvent : Pointer to FB_EventTrigger
VAR_INPUT
	nIndex:UINT;
END_VAR
IF nIndex >=0 AND nIndex <nWriteIndex THEN
	GetEvent:= aFaultsToCheck[nIndex];
ELSE
	//TODO-NIKO error gracefully
END_IF
END_METHOD

METHOD PUBLIC GetFirstActiveEvent : Pointer TO FB_EventTrigger
VAR_INPUT
END_VAR
//FOR nIdx := LOWER_BOUND(aFaultsToCheck,1) TO UPPER_BOUND(aFaultsToCheck,1) DO

FOR nIdx := 0 TO nWriteIndex-1 DO
	//IF(aFaultsToCheck[nIdx]^.GetState()) THEN
	//	GetFirstActiveEvent:=aFaultsToCheck[nIdx];
	//	EXIT;
	//END_IF
END_FOR;
END_METHOD

METHOD GetTotalEventCount : UINT
VAR_INPUT
END_VAR
GetTotalEventCount:=nWriteIndex;
END_METHOD

METHOD Update
VAR_INPUT
END_VAR
//FOR nIdx := LOWER_BOUND(aFaultsToCheck,1) TO UPPER_BOUND(aFaultsToCheck,1) DO


FOR nIdx := 0 TO nWriteIndex-1 DO
(*	ADSLOGSTR(
	msgCtrlMask := ADSLOG_MSGTYPE_HINT, 
	msgFmtStr   := 'IndexWas %s', 
	strArg      := TO_STRING(nIDX)
	//TODO-NIKO DELETE DEBUG CODE COMMENT
	
);  *)
//aFaultsToCheck[nIdx]^.Update();
END_FOR;
END_METHOD

END_FUNCTION_BLOCK

// ---- FaultChecker/FB_EventTrigger.TcPOU
FUNCTION_BLOCK FB_EventTrigger
VAR_INPUT
	
END_VAR
VAR_OUTPUT
END_VAR
VAR
	bTriggered:BOOL;
	
	aTriggerData : ARRAY [0..1000] OF TriggerData ;
	aTriggerSettings : ARRAY [0..1000] OF TriggerSettings ;
	myClass : GUID;
	fbTcMessage		: FB_TcMessage;
	fbSource		: FB_TcSourceInfo;
	
	//selfSource: FB_TcSourceInfo;
END_VAR

METHOD PUBLIC Configure
VAR_INPUT
	nEventID : UDINT;
	stTriggerSettings : TriggerSettings;
END_VAR
aTriggerSettings[nEventID]:=stTriggerSettings;
END_METHOD

//FB_Init is always available implicitly and it is used primarily for initialization.
//The return value is not evaluated. For a specific influence, you can also declare the
//methods explicitly and provide additional code there with the standard initialization
//code. You can evaluate the return value.
METHOD FB_Init: BOOL
VAR_INPUT
    bInitRetains: BOOL; // TRUE: the retain variables are initialized (reset warm / reset cold)
    bInCopyCode: BOOL;  // TRUE: the instance will be copied to the copy code afterward (online change)   
	eventClass : GUID;
END_VAR
myClass:=eventClass;
END_METHOD

METHOD PUBLIC GetState : BOOL
VAR_INPUT
	nEventID : UDINT;
END_VAR
GetState:=aTriggerData[nEventID].bTriggered;
END_METHOD

METHOD PUBLIC placeholder
VAR_INPUT
		nEventEntry: TcEventEntry;
	nEventID: UDINT:=0;

	bTrigger: BOOL;
	sSource: STRING :=__POUNAME();
	nI : INT :=0;
	nJ : INT :=0;
	sK : STRING :='';
	eSeverity :TcEventSeverity:=TcEventSeverity.Verbose;
END_VAR
END_METHOD

METHOD PUBLIC Reset
VAR_INPUT
	nEventID : UDINT;
END_VAR
aTriggerData[nEventID].bTriggered:=FALSE;
aTriggerData[nEventID].nActivationCount:=0;
END_METHOD

METHOD PUBLIC Trigger
VAR_INPUT
	nEventID: UDINT;
	bTrigger: BOOL;
	sSource: STRING :=__POUNAME();
	arg1 : STRING :='';
	arg2 : STRING :='';
	arg3 : STRING :='';
	eSeverity :TcEventSeverity:=TcEventSeverity.Verbose;
END_VAR
VAR
	string1 :STRING;
string2 :STRING;
string3:STRING;
END_VAR
fbSource.sName:=sSource;
string1:=TO_STRING(arg1);
string2:=TO_STRING(arg2);
string3:=TO_STRING(arg3);


IF aTriggerSettings[nEventID].tDebounceTime > T#0MS THEN
	aTriggerData[nEventID].timerDebounceTimer(IN:= bTrigger, PT := aTriggerSettings[nEventID].tDebounceTime);
	aTriggerData[nEventID].GetEventTrigger(CLK:=aTriggerData[nEventID].timerDebounceTimer.Q);
ELSE
	aTriggerData[nEventID].GetEventTrigger(CLK:=bTrigger);
END_IF

IF aTriggerData[nEventID].GetEventTrigger.Q THEN
	aTriggerData[nEventID].nActivationCount := aTriggerData[nEventID].nActivationCount +1;
END_IF



IF(aTriggerData[nEventID].nActivationCount >= aTriggerSettings[nEventID].nActivationThreshold) THEN
	aTriggerData[nEventID].bTriggered :=TRUE;
ELSE	
	aTriggerData[nEventID].bTriggered:=FALSE;
END_IF

IF aTriggerSettings[nEventID].bAutoResetCount AND bTrigger = FALSE THEN
	aTriggerData[nEventID].nActivationCount :=0;
END_IF




aTriggerData[nEventID].SendEventTrigger(CLK:=aTriggerData[nEventID].bTriggered);

IF aTriggerData[nEventID].SendEventTrigger.Q THEN
	IF(aTriggerSettings[nEventID].eEventType = E_EventType.Message) THEN
		fbTcMessage.Create(eventClass:=myClass, nEventID:= TO_UDINT(nEventID), eSeverity:=eSeverity ,ipSourceInfo:=fbSource);
		fbTcMessage.ipArguments.Clear();
		fbTcMessage.ipArguments.AddUDInt(TO_UDINT(nEventID));
		fbTcMessage.ipArguments.AddString(string1);
		fbTcMessage.ipArguments.AddString(string2);
		fbTcMessage.ipArguments.AddString(string3);
		fbTcMessage.Send(0);
	
	ELSE
		fbTcMessage.Create(eventClass:=TC_EVENT_CLASSES.TestEventClass, nEventID:= TO_UDINT(nEventID), eSeverity:=eSeverity ,ipSourceInfo:=fbSource);
		fbTcMessage.ipArguments.Clear();
		fbTcMessage.ipArguments.AddUDInt(TO_UDINT(nEventID));
		fbTcMessage.ipArguments.AddString(string1);
		fbTcMessage.ipArguments.AddString(string2);
		fbTcMessage.ipArguments.AddString(string3);
		fbTcMessage.Send(0);
	END_IF
END_IF
END_METHOD

METHOD PUBLIC TriggerEvent//A wrapper provided for convience. Only differs From Trigger in the data type. 
VAR_INPUT
	nEventEntry: TcEventEntry;
	bTrigger: BOOL;
	sSource: STRING :=__POUNAME();
	arg1 : STRING :='';
	arg2 : STRING :='';
	arg3 : STRING :='';
	eSeverity :TcEventSeverity:=TcEventSeverity.Verbose;
END_VAR
Trigger(nEventID:=nEventEntry.nEventId,bTrigger,sSource,arg1,arg2,arg3,eSeverity);
END_METHOD

END_FUNCTION_BLOCK

// ---- FaultChecker/TC_EventSeverityToString.TcPOU
FUNCTION TC_EventSeverityToString : STRING
VAR_INPUT
	eSeverity: TcEventSeverity;
END_VAR
VAR
	sSeverity:STRING;
END_VAR

CASE eSeverity OF
    TcEventSeverity.Verbose:
        sSeverity := 'Verbose';
    TcEventSeverity.Info:
        sSeverity := 'Info';
    TcEventSeverity.Warning:
        sSeverity := 'Warning';
    TcEventSeverity.Error:
        sSeverity := 'Error';
    TcEventSeverity.Critical:
        sSeverity := 'Critical';
ELSE
    sSeverity := 'Unknown';
END_CASE

TC_EventSeverityToString := sSeverity;

END_FUNCTION
